(* CODESYS project IndraLogic.project

Project tree, tasks and I/O mapping:
  IndraMotionMlc1 : IndraMotion MLC L25, Bosch Rexroth AG, order no. R911171363, version 14.20.34.0
    application Application
      task PlcTask (cyclic, interval 10 ms, priority 5, watchdog 100 ms x 2) calls PlcProg
      global variables UserVarGlobal
      Symbols
      program PlcProg [ST]
      visualisation Visualization
      global variables MlcVarGlobal
      visualisation TestFrame
      image pool ImagePool
      program Datensimulator [ST]
      program Visualisierungssteuerung [ST]
      function block GenAngleTest [ST]
    Inline_I_O : Inline I/O, Bosch Rexroth AG, version 12.8.2.0
    Sercos_III_Master : SercosIII Master, Rexroth, order no. 1, version 14.6.0.0
  text list GlobalTextList
  5ce3da45-db07-42e7-a21c-a00fff4ed8f6|C:\Users\Kun\Desktop\Uni\Automatisierungstechnik\ProjektaufgabeAT\Overlay.png
*)

// IndraMotionMlc1/Application/UserVarGlobal
{attribute 'qualified_only'}
VAR_GLOBAL
END_VAR

// IndraMotionMlc1/Application/MlcVarGlobal
(* Automatically generated code by XLC/MLC. *)
(* Please don't edit, the code will be overwritten. For usercode use UserVarGlobal! *)
{attribute 'linkalways'}
{attribute 'analysis' := '-33'}
VAR_GLOBAL CONSTANT

(*Probe 001*)
TouchProbe001: TOUCHPROBE_REF :=(CntrlNo:=LOCAL_CNTRL,TouchProbeNo:=TOUCHPROBE_1);

(*Probe 002*)
TouchProbe002: TOUCHPROBE_REF :=(CntrlNo:=LOCAL_CNTRL,TouchProbeNo:=TOUCHPROBE_2);

(*Probe 003*)
TouchProbe003: TOUCHPROBE_REF :=(CntrlNo:=LOCAL_CNTRL,TouchProbeNo:=TOUCHPROBE_3);

(*Probe 004*)
TouchProbe004: TOUCHPROBE_REF :=(CntrlNo:=LOCAL_CNTRL,TouchProbeNo:=TOUCHPROBE_4);

(*Probe 005*)
TouchProbe005: TOUCHPROBE_REF :=(CntrlNo:=LOCAL_CNTRL,TouchProbeNo:=TOUCHPROBE_5);

(*Probe 006*)
TouchProbe006: TOUCHPROBE_REF :=(CntrlNo:=LOCAL_CNTRL,TouchProbeNo:=TOUCHPROBE_6);

(*Probe 007*)
TouchProbe007: TOUCHPROBE_REF :=(CntrlNo:=LOCAL_CNTRL,TouchProbeNo:=TOUCHPROBE_7);

(*Probe 008*)
TouchProbe008: TOUCHPROBE_REF :=(CntrlNo:=LOCAL_CNTRL,TouchProbeNo:=TOUCHPROBE_8);

(*Probe 009*)
TouchProbe009: TOUCHPROBE_REF :=(CntrlNo:=LOCAL_CNTRL,TouchProbeNo:=TOUCHPROBE_9);

(*Probe 010*)
TouchProbe010: TOUCHPROBE_REF :=(CntrlNo:=LOCAL_CNTRL,TouchProbeNo:=TOUCHPROBE_10);

(*Probe 011*)
TouchProbe011: TOUCHPROBE_REF :=(CntrlNo:=LOCAL_CNTRL,TouchProbeNo:=TOUCHPROBE_11);

(*Probe 012*)
TouchProbe012: TOUCHPROBE_REF :=(CntrlNo:=LOCAL_CNTRL,TouchProbeNo:=TOUCHPROBE_12);

(*Probe 013*)
TouchProbe013: TOUCHPROBE_REF :=(CntrlNo:=LOCAL_CNTRL,TouchProbeNo:=TOUCHPROBE_13);

(*Probe 014*)
TouchProbe014: TOUCHPROBE_REF :=(CntrlNo:=LOCAL_CNTRL,TouchProbeNo:=TOUCHPROBE_14);

(*Probe 015*)
TouchProbe015: TOUCHPROBE_REF :=(CntrlNo:=LOCAL_CNTRL,TouchProbeNo:=TOUCHPROBE_15);

(*Probe 016*)
TouchProbe016: TOUCHPROBE_REF :=(CntrlNo:=LOCAL_CNTRL,TouchProbeNo:=TOUCHPROBE_16);

(*Probe 017*)
TouchProbe017: TOUCHPROBE_REF :=(CntrlNo:=LOCAL_CNTRL,TouchProbeNo:=TOUCHPROBE_17);

(*Probe 018*)
TouchProbe018: TOUCHPROBE_REF :=(CntrlNo:=LOCAL_CNTRL,TouchProbeNo:=TOUCHPROBE_18);

(*Probe 019*)
TouchProbe019: TOUCHPROBE_REF :=(CntrlNo:=LOCAL_CNTRL,TouchProbeNo:=TOUCHPROBE_19);

(*Probe 020*)
TouchProbe020: TOUCHPROBE_REF :=(CntrlNo:=LOCAL_CNTRL,TouchProbeNo:=TOUCHPROBE_20);

(*Probe 021*)
TouchProbe021: TOUCHPROBE_REF :=(CntrlNo:=LOCAL_CNTRL,TouchProbeNo:=TOUCHPROBE_21);

(*Probe 022*)
TouchProbe022: TOUCHPROBE_REF :=(CntrlNo:=LOCAL_CNTRL,TouchProbeNo:=TOUCHPROBE_22);

(*Probe 023*)
TouchProbe023: TOUCHPROBE_REF :=(CntrlNo:=LOCAL_CNTRL,TouchProbeNo:=TOUCHPROBE_23);

(*Probe 024*)
TouchProbe024: TOUCHPROBE_REF :=(CntrlNo:=LOCAL_CNTRL,TouchProbeNo:=TOUCHPROBE_24);

(*Probe 025*)
TouchProbe025: TOUCHPROBE_REF :=(CntrlNo:=LOCAL_CNTRL,TouchProbeNo:=TOUCHPROBE_25);

(*Probe 026*)
TouchProbe026: TOUCHPROBE_REF :=(CntrlNo:=LOCAL_CNTRL,TouchProbeNo:=TOUCHPROBE_26);

(*Probe 027*)
TouchProbe027: TOUCHPROBE_REF :=(CntrlNo:=LOCAL_CNTRL,TouchProbeNo:=TOUCHPROBE_27);

(*Probe 028*)
TouchProbe028: TOUCHPROBE_REF :=(CntrlNo:=LOCAL_CNTRL,TouchProbeNo:=TOUCHPROBE_28);

(*Probe 029*)
TouchProbe029: TOUCHPROBE_REF :=(CntrlNo:=LOCAL_CNTRL,TouchProbeNo:=TOUCHPROBE_29);

(*Probe 030*)
TouchProbe030: TOUCHPROBE_REF :=(CntrlNo:=LOCAL_CNTRL,TouchProbeNo:=TOUCHPROBE_30);

(*Probe 031*)
TouchProbe031: TOUCHPROBE_REF :=(CntrlNo:=LOCAL_CNTRL,TouchProbeNo:=TOUCHPROBE_31);

(*Probe 032*)
TouchProbe032: TOUCHPROBE_REF :=(CntrlNo:=LOCAL_CNTRL,TouchProbeNo:=TOUCHPROBE_32);

(*Probe 033*)
TouchProbe033: TOUCHPROBE_REF :=(CntrlNo:=LOCAL_CNTRL,TouchProbeNo:=TOUCHPROBE_33);

(*Probe 034*)
TouchProbe034: TOUCHPROBE_REF :=(CntrlNo:=LOCAL_CNTRL,TouchProbeNo:=TOUCHPROBE_34);

(*Probe 035*)
TouchProbe035: TOUCHPROBE_REF :=(CntrlNo:=LOCAL_CNTRL,TouchProbeNo:=TOUCHPROBE_35);

(*Probe 036*)
TouchProbe036: TOUCHPROBE_REF :=(CntrlNo:=LOCAL_CNTRL,TouchProbeNo:=TOUCHPROBE_36);

(*Probe 037*)
TouchProbe037: TOUCHPROBE_REF :=(CntrlNo:=LOCAL_CNTRL,TouchProbeNo:=TOUCHPROBE_37);

(*Probe 038*)
TouchProbe038: TOUCHPROBE_REF :=(CntrlNo:=LOCAL_CNTRL,TouchProbeNo:=TOUCHPROBE_38);

(*Probe 039*)
TouchProbe039: TOUCHPROBE_REF :=(CntrlNo:=LOCAL_CNTRL,TouchProbeNo:=TOUCHPROBE_39);

(*Probe 040*)
TouchProbe040: TOUCHPROBE_REF :=(CntrlNo:=LOCAL_CNTRL,TouchProbeNo:=TOUCHPROBE_40);

(*Probe 041*)
TouchProbe041: TOUCHPROBE_REF :=(CntrlNo:=LOCAL_CNTRL,TouchProbeNo:=TOUCHPROBE_41);

(*Probe 042*)
TouchProbe042: TOUCHPROBE_REF :=(CntrlNo:=LOCAL_CNTRL,TouchProbeNo:=TOUCHPROBE_42);

(*Probe 043*)
TouchProbe043: TOUCHPROBE_REF :=(CntrlNo:=LOCAL_CNTRL,TouchProbeNo:=TOUCHPROBE_43);

(*Probe 044*)
TouchProbe044: TOUCHPROBE_REF :=(CntrlNo:=LOCAL_CNTRL,TouchProbeNo:=TOUCHPROBE_44);

(*Probe 045*)
TouchProbe045: TOUCHPROBE_REF :=(CntrlNo:=LOCAL_CNTRL,TouchProbeNo:=TOUCHPROBE_45);

(*Probe 046*)
TouchProbe046: TOUCHPROBE_REF :=(CntrlNo:=LOCAL_CNTRL,TouchProbeNo:=TOUCHPROBE_46);

(*Probe 047*)
TouchProbe047: TOUCHPROBE_REF :=(CntrlNo:=LOCAL_CNTRL,TouchProbeNo:=TOUCHPROBE_47);

(*Probe 048*)
TouchProbe048: TOUCHPROBE_REF :=(CntrlNo:=LOCAL_CNTRL,TouchProbeNo:=TOUCHPROBE_48);

(*Probe 049*)
TouchProbe049: TOUCHPROBE_REF :=(CntrlNo:=LOCAL_CNTRL,TouchProbeNo:=TOUCHPROBE_49);

(*Probe 050*)
TouchProbe050: TOUCHPROBE_REF :=(CntrlNo:=LOCAL_CNTRL,TouchProbeNo:=TOUCHPROBE_50);

(*Probe 051*)
TouchProbe051: TOUCHPROBE_REF :=(CntrlNo:=LOCAL_CNTRL,TouchProbeNo:=TOUCHPROBE_51);

(*Probe 052*)
TouchProbe052: TOUCHPROBE_REF :=(CntrlNo:=LOCAL_CNTRL,TouchProbeNo:=TOUCHPROBE_52);

(*Probe 053*)
TouchProbe053: TOUCHPROBE_REF :=(CntrlNo:=LOCAL_CNTRL,TouchProbeNo:=TOUCHPROBE_53);

(*Probe 054*)
TouchProbe054: TOUCHPROBE_REF :=(CntrlNo:=LOCAL_CNTRL,TouchProbeNo:=TOUCHPROBE_54);

(*Probe 055*)
TouchProbe055: TOUCHPROBE_REF :=(CntrlNo:=LOCAL_CNTRL,TouchProbeNo:=TOUCHPROBE_55);

(*Probe 056*)
TouchProbe056: TOUCHPROBE_REF :=(CntrlNo:=LOCAL_CNTRL,TouchProbeNo:=TOUCHPROBE_56);

(*Probe 057*)
TouchProbe057: TOUCHPROBE_REF :=(CntrlNo:=LOCAL_CNTRL,TouchProbeNo:=TOUCHPROBE_57);

(*Probe 058*)
TouchProbe058: TOUCHPROBE_REF :=(CntrlNo:=LOCAL_CNTRL,TouchProbeNo:=TOUCHPROBE_58);

(*Probe 059*)
TouchProbe059: TOUCHPROBE_REF :=(CntrlNo:=LOCAL_CNTRL,TouchProbeNo:=TOUCHPROBE_59);

(*Probe 060*)
TouchProbe060: TOUCHPROBE_REF :=(CntrlNo:=LOCAL_CNTRL,TouchProbeNo:=TOUCHPROBE_60);

(*Probe 061*)
TouchProbe061: TOUCHPROBE_REF :=(CntrlNo:=LOCAL_CNTRL,TouchProbeNo:=TOUCHPROBE_61);

(*Probe 062*)
TouchProbe062: TOUCHPROBE_REF :=(CntrlNo:=LOCAL_CNTRL,TouchProbeNo:=TOUCHPROBE_62);

(*Probe 063*)
TouchProbe063: TOUCHPROBE_REF :=(CntrlNo:=LOCAL_CNTRL,TouchProbeNo:=TOUCHPROBE_63);

(*Probe 064*)
TouchProbe064: TOUCHPROBE_REF :=(CntrlNo:=LOCAL_CNTRL,TouchProbeNo:=TOUCHPROBE_64);

(*Probe 065*)
TouchProbe065: TOUCHPROBE_REF :=(CntrlNo:=LOCAL_CNTRL,TouchProbeNo:=TOUCHPROBE_65);

(*Probe 066*)
TouchProbe066: TOUCHPROBE_REF :=(CntrlNo:=LOCAL_CNTRL,TouchProbeNo:=TOUCHPROBE_66);

(*Probe 067*)
TouchProbe067: TOUCHPROBE_REF :=(CntrlNo:=LOCAL_CNTRL,TouchProbeNo:=TOUCHPROBE_67);

(*Probe 068*)
TouchProbe068: TOUCHPROBE_REF :=(CntrlNo:=LOCAL_CNTRL,TouchProbeNo:=TOUCHPROBE_68);

(*Probe 069*)
TouchProbe069: TOUCHPROBE_REF :=(CntrlNo:=LOCAL_CNTRL,TouchProbeNo:=TOUCHPROBE_69);

(*Probe 070*)
TouchProbe070: TOUCHPROBE_REF :=(CntrlNo:=LOCAL_CNTRL,TouchProbeNo:=TOUCHPROBE_70);

(*Probe 071*)
TouchProbe071: TOUCHPROBE_REF :=(CntrlNo:=LOCAL_CNTRL,TouchProbeNo:=TOUCHPROBE_71);

(*Probe 072*)
TouchProbe072: TOUCHPROBE_REF :=(CntrlNo:=LOCAL_CNTRL,TouchProbeNo:=TOUCHPROBE_72);

(*Probe 073*)
TouchProbe073: TOUCHPROBE_REF :=(CntrlNo:=LOCAL_CNTRL,TouchProbeNo:=TOUCHPROBE_73);

(*Probe 074*)
TouchProbe074: TOUCHPROBE_REF :=(CntrlNo:=LOCAL_CNTRL,TouchProbeNo:=TOUCHPROBE_74);

(*Probe 075*)
TouchProbe075: TOUCHPROBE_REF :=(CntrlNo:=LOCAL_CNTRL,TouchProbeNo:=TOUCHPROBE_75);

(*Probe 076*)
TouchProbe076: TOUCHPROBE_REF :=(CntrlNo:=LOCAL_CNTRL,TouchProbeNo:=TOUCHPROBE_76);

(*Probe 077*)
TouchProbe077: TOUCHPROBE_REF :=(CntrlNo:=LOCAL_CNTRL,TouchProbeNo:=TOUCHPROBE_77);

(*Probe 078*)
TouchProbe078: TOUCHPROBE_REF :=(CntrlNo:=LOCAL_CNTRL,TouchProbeNo:=TOUCHPROBE_78);

(*Probe 079*)
TouchProbe079: TOUCHPROBE_REF :=(CntrlNo:=LOCAL_CNTRL,TouchProbeNo:=TOUCHPROBE_79);

(*Probe 080*)
TouchProbe080: TOUCHPROBE_REF :=(CntrlNo:=LOCAL_CNTRL,TouchProbeNo:=TOUCHPROBE_80);

(*Probe 081*)
TouchProbe081: TOUCHPROBE_REF :=(CntrlNo:=LOCAL_CNTRL,TouchProbeNo:=TOUCHPROBE_81);

(*Probe 082*)
TouchProbe082: TOUCHPROBE_REF :=(CntrlNo:=LOCAL_CNTRL,TouchProbeNo:=TOUCHPROBE_82);

(*Probe 083*)
TouchProbe083: TOUCHPROBE_REF :=(CntrlNo:=LOCAL_CNTRL,TouchProbeNo:=TOUCHPROBE_83);

(*Probe 084*)
TouchProbe084: TOUCHPROBE_REF :=(CntrlNo:=LOCAL_CNTRL,TouchProbeNo:=TOUCHPROBE_84);

(*Probe 085*)
TouchProbe085: TOUCHPROBE_REF :=(CntrlNo:=LOCAL_CNTRL,TouchProbeNo:=TOUCHPROBE_85);

(*Probe 086*)
TouchProbe086: TOUCHPROBE_REF :=(CntrlNo:=LOCAL_CNTRL,TouchProbeNo:=TOUCHPROBE_86);

(*Probe 087*)
TouchProbe087: TOUCHPROBE_REF :=(CntrlNo:=LOCAL_CNTRL,TouchProbeNo:=TOUCHPROBE_87);

(*Probe 088*)
TouchProbe088: TOUCHPROBE_REF :=(CntrlNo:=LOCAL_CNTRL,TouchProbeNo:=TOUCHPROBE_88);

(*Probe 089*)
TouchProbe089: TOUCHPROBE_REF :=(CntrlNo:=LOCAL_CNTRL,TouchProbeNo:=TOUCHPROBE_89);

(*Probe 090*)
TouchProbe090: TOUCHPROBE_REF :=(CntrlNo:=LOCAL_CNTRL,TouchProbeNo:=TOUCHPROBE_90);

(*Probe 091*)
TouchProbe091: TOUCHPROBE_REF :=(CntrlNo:=LOCAL_CNTRL,TouchProbeNo:=TOUCHPROBE_91);

(*Probe 092*)
TouchProbe092: TOUCHPROBE_REF :=(CntrlNo:=LOCAL_CNTRL,TouchProbeNo:=TOUCHPROBE_92);

(*Probe 093*)
TouchProbe093: TOUCHPROBE_REF :=(CntrlNo:=LOCAL_CNTRL,TouchProbeNo:=TOUCHPROBE_93);

(*Probe 094*)
TouchProbe094: TOUCHPROBE_REF :=(CntrlNo:=LOCAL_CNTRL,TouchProbeNo:=TOUCHPROBE_94);

(*Probe 095*)
TouchProbe095: TOUCHPROBE_REF :=(CntrlNo:=LOCAL_CNTRL,TouchProbeNo:=TOUCHPROBE_95);

(*Probe 096*)
TouchProbe096: TOUCHPROBE_REF :=(CntrlNo:=LOCAL_CNTRL,TouchProbeNo:=TOUCHPROBE_96);

(*Probe 097*)
TouchProbe097: TOUCHPROBE_REF :=(CntrlNo:=LOCAL_CNTRL,TouchProbeNo:=TOUCHPROBE_97);

(*Probe 098*)
TouchProbe098: TOUCHPROBE_REF :=(CntrlNo:=LOCAL_CNTRL,TouchProbeNo:=TOUCHPROBE_98);

(*Probe 099*)
TouchProbe099: TOUCHPROBE_REF :=(CntrlNo:=LOCAL_CNTRL,TouchProbeNo:=TOUCHPROBE_99);

(*Probe 100*)
TouchProbe100: TOUCHPROBE_REF :=(CntrlNo:=LOCAL_CNTRL,TouchProbeNo:=TOUCHPROBE_100);

END_VAR

// IndraMotionMlc1/Application/PlcProg
PROGRAM PlcProg
VAR
	rPitch 		: 	SINT;
	rRoll 		: 	REAL;
	height		:	REAL;
	speed		:	UINT	:=	10;
	climbRate	:	REAL;
	rDirection	:	REAL;
	steps		:	LINT;
	bEnableTest	:	BOOL 	:= TRUE;
	rollTest	:	GenAngleTest;
	test		:	REAL;
END_VAR

VAR CONSTANT
	timestep	:	INT		:=	5;	// Timestep
	
END_VAR

rollTest(benable:=bEnableTest,startAngle:=-20.0,finalAngle:=20.0,sweepTime:=500);
rRoll := rollTest.Angle/1;
IF (rollTest.active = FALSE) THEN
	rRoll := 0;
END_IF

END_PROGRAM

// IndraMotionMlc1/Application/GenAngleTest
FUNCTION_BLOCK GenAngleTest
VAR_INPUT
	bEnable			: BOOL;
	startAngle		: REAL;
	finalAngle		: REAL;
	sweepTime		: INT;	//Sweeptime in cycles
END_VAR
VAR_OUTPUT
	Angle			: REAL;
	active			: BOOL;
END_VAR
VAR
	internalTimer	: INT;
	angleInc		: REAL;
	bFirstSweep		: BOOL := TRUE;	// Winkel soll einmal in beide Richtugnen veränder werden
END_VAR

angleInc := -(startAngle-finalAngle)/sweepTime;
IF (bEnable AND internalTimer < sweepTime AND bFirstSweep) THEN
	Angle := startAngle + angleInc * internalTimer;
	internalTimer := internalTimer + 1;
	active := TRUE;
ELSIF (internalTimer = sweepTime) THEN
	bFirstSweep := FALSE;
END_IF
IF (bFirstSweep = FALSE AND internalTimer > 0) THEN
	Angle := finalAngle + angleInc * (internalTimer-sweepTime);
	internalTimer := internalTimer - 1;
ELSIF (bFirstSweep = FALSE AND internalTimer = 0) THEN
	active := FALSE;
END_IF
IF (bEnable = FALSE) THEN
	Angle := 0;
	internalTimer := 0;
	angleInc := 0;
	bFirstSweep := TRUE;
	active := FALSE;
END_IF

END_FUNCTION_BLOCK

// IndraMotionMlc1/Application/Datensimulator
PROGRAM Datensimulator
VAR
END_VAR

END_PROGRAM

// IndraMotionMlc1/Application/Visualisierungssteuerung
PROGRAM Visualisierungssteuerung
VAR
END_VAR

END_PROGRAM

// IndraMotionMlc1/Application/Visualization
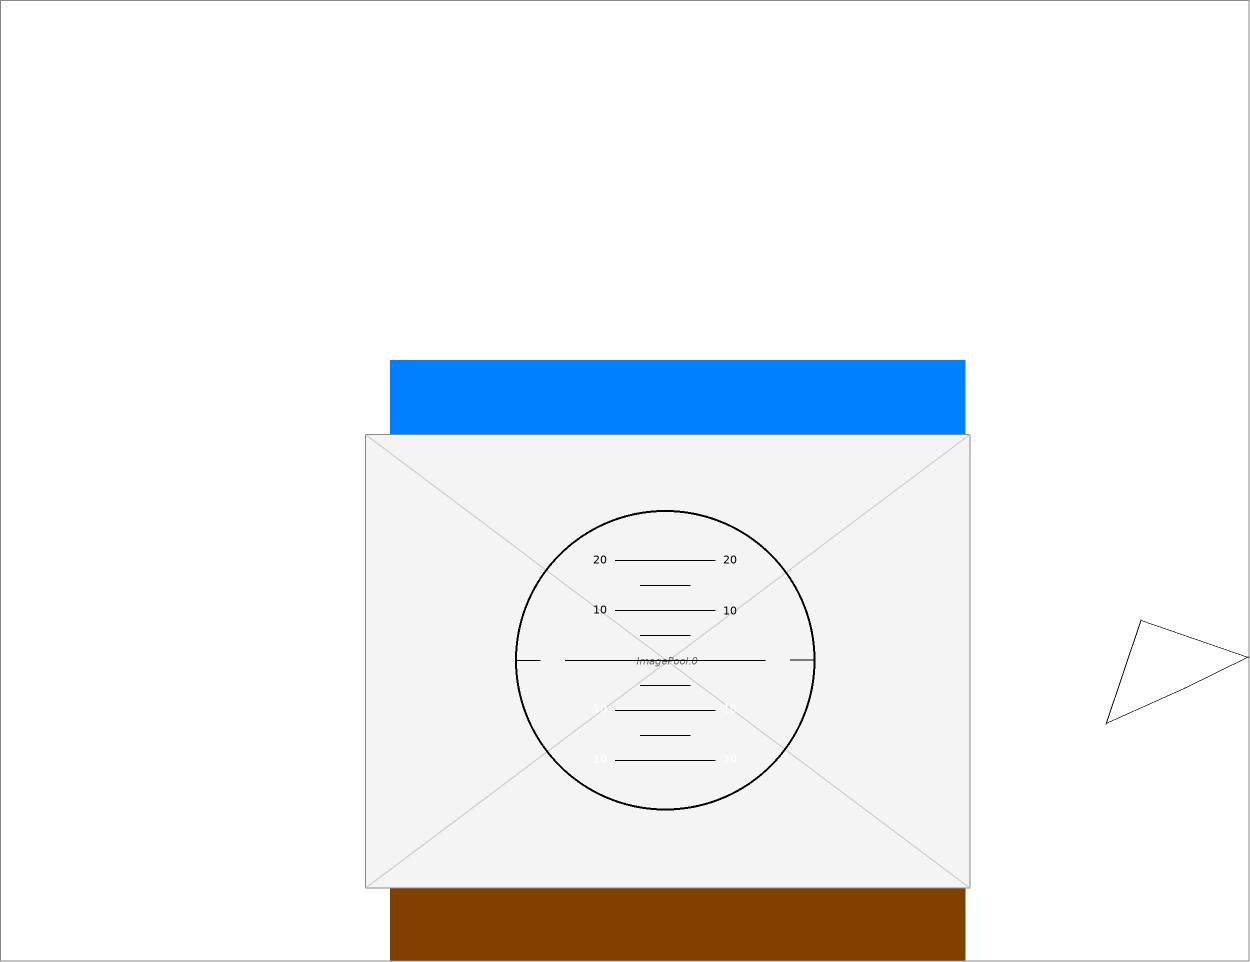
VISUALIZATION Visualization  // 1250x962
    Rectangle (390,660 575x300)
        p2858320360: PlcProg.rRoll
    Rectangle (390,360 575x300)
        p2858320360: PlcProg.rRoll
    Image (365,434 605x454), image: ImagePool.0
    Ellipse (515,510 300x300)
        p2858320360: PlcProg.rRoll
    Line (565,660) (765,660)
        p2858320360: PlcProg.rRoll
    Line (640,635) (690,635)
        p2858320360: PlcProg.rRoll
    Line (615,610) (715,610)
        p2858320360: PlcProg.rRoll
    Line (640,585) (690,585)
        p2858320360: PlcProg.rRoll
    Line (640,685) (690,685)
        p2858320360: PlcProg.rRoll
    Line (615,710) (715,710)
        p2858320360: PlcProg.rRoll
    Line (640,735) (690,735)
        p2858320360: PlcProg.rRoll
    Line (615,560) (715,560)
        p2858320360: PlcProg.rRoll
    Line (615,760) (715,760)
        p2858320360: PlcProg.rRoll
    Line (815,660) (790,660)
    Line (515,660) (540,660)
    Rectangle (715,597 30x28), "10"
        p2858320360: PlcProg.rRoll
    Rectangle (715,545 30x30), "20"
        p2858320360: PlcProg.rRoll
    Rectangle (585,595 30x30), "10"
        p2858320360: PlcProg.rRoll
    Rectangle (585,545 30x30), "20"
        p2858320360: PlcProg.rRoll
    Polyline (1106,724) (1141,620) (1248,657) (1185,688) (1107,723)
    Rectangle (715,695 30x28), "10"
        p2858320360: PlcProg.rRoll
    Rectangle (585,695 30x28), "10"
        p2858320360: PlcProg.rRoll
    Rectangle (715,745 30x28), "10"
        p2858320360: PlcProg.rRoll
    Rectangle (585,745 30x28), "10"
        p2858320360: PlcProg.rRoll
END_VISUALIZATION

// IndraMotionMlc1/Application/TestFrame
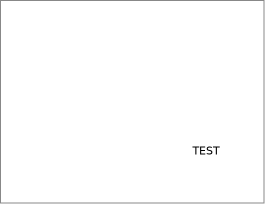
VISUALIZATION TestFrame  // 265x204
    Label (149,100 114x102), "TEST"
END_VISUALIZATION
